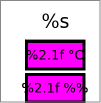
VISUALIZATION Obj_THT_Field  // 101x103
VAR_INPUT;
	rTempValue : REAL;
	rHumValue : REAL;
	bTempLimitAlarm : BOOL;
	bHumLimitAlarm : BOOL;
	bTempFailed : BOOL;
	bHumFailed : BOOL;
	bTempOffline : BOOL;
	bHumOffline : BOOL;
	bTempExcluded : BOOL;
	bHumExcluded : BOOL;
	bDeactivateDialog : BOOL;
END_VAR
    Rectangle (10,8 91x27), "%s", text variable: sIndex
    Group (25,39 60x64)
        Rectangle (0,34 60x30), "%2.1f %%", text variable: rHumValue, colour toggle: bHumLimitAlarm
        Rectangle (0,1 60x30), "%2.1f °C", text variable: rTempValue, colour toggle: bTempLimitAlarm
        Rectangle (0,0 60x30), "%2.1f °C", text variable: rTempValue, invisible if: NOT bTempExcluded
        Rectangle (0,1 60x30), "OoR", invisible if: NOT bTempFailed
        Rectangle (0,34 60x30), "%2.1f %%", text variable: rHumValue, invisible if: not bHumExcluded
        Rectangle (0,34 60x30), "OoR", invisible if: Not bHumFailed
        Line (60,30) (0,1), invisible if: not bTempExcluded
        Line (60,64) (0,35), invisible if: not bHumExcluded
        Rectangle (0,1 60x30), "%2.1f °C", text variable: rTempValue, invisible if: NOT bTempOffline
        Rectangle (0,34 60x30), "%2.1f %%", text variable: rHumValue, invisible if: NOT bHumOffline
END_VISUALIZATION

(* stored: Version 1.1.0.1, ProductVersion 3.1.4024.12
   Visu Obj_THT_Field: Id {e2df1fda-7525-473b-9342-cc9c45a09a09} *)
